{attribute 'qualified_only'}
{attribute 'strict'}
TYPE E_STREAMSEEKTYPE :
(
	Origin := 0,
	Current,
	End
);
END_TYPE

(* stored: Version 1.1.0.1, ProductVersion 3.1.4019.2
   DUT E_STREAMSEEKTYPE: Id {8af1dfd2-3bc9-411e-815a-f28cc258cce5} *)
